(* CoDeSys 2.3.10.0 project: BC_068364(3.222)-prg__2014.10.23.prx *)
(* Libraries: standard.lbx 5.12.03 07:02:30, TcBaseBCxx50.lbx 29.3.07 05:21:36, TcSystemBCxx50.lbx*11.2.10 13:45:50, TcpIp.lib 9.1.14 12:33:22 *)

(* Task configuration *)
TASK Standard (PRIORITY := 0, INTERVAL := T#20ms);
	ADS_block();
	MAIN
END_TASK

(* Global variable list: Global_Variables *)
VAR_GLOBAL
	IN_DGU AT %I* : BOOL; (*сигнал старта дгу / IN1 на MU1.6 KL1702*)
	IN_TEMP AT %I* : INT; (*температура воздуха в гараже / IN1 на MU1.3 KL4002*)
	IN_CO2 AT %I* : INT; (*содержание СО2 в гараже / IN2 на MU1.3 KL4002*)
	OUT_START_V1 AT %Q* : BOOL; (*старт пускателя В-1 / IN1 на MU1.1 KM2642*)
	OUT_START_V2 AT %Q* : BOOL; (*старт пускателя В-2 / IN2 на MU1.1 KM2642*)
	OUT_START_V3 AT %Q* : BOOL; (*старт вентилятора в туалете Николая В-3 / IN1 на MU1.2 KM2642*)
	OUT_OUTPUT_V1 AT %Q* : INT; (*производительность В-1 / OUT1 на MU1.3 KL4002*)
	OUT_OUTPUT_V2 AT %Q* : INT; (*производительность В-2 / OUT2 на MU1.3 KL4002*)
	Ads_Udp_send_Stack : ARRAY [1..7] OF INT; (*информационный массив для передачи по ADS*)
	Ads_Udp_receive_Stack : ARRAY [1..7] OF INT; (*информационный массив для получения по ADS*)
	Ads_Udp_empty_Stack : ARRAY [1..7] OF INT := 0;
	Garage_OG10_11: BOOL := FALSE;
	Garage AT %MB10 : BOOL;

	var1 : BOOL;
	var2: BOOL;
	var3 : BOOL;
END_VAR

(* Global variable list: TwinCAT_Configuration *)
(* Generated automatically by TwinCAT - (read only) *)
VAR_CONFIG
	.IN_DGU AT %IX8.0 : BOOL;	(*  ~ {LinkedWith:TIID^Device 2 (BX-BK)^BX KBus-Device^Term 7 (KL1702)^Channel 1^Input} *)
	.IN_TEMP AT %IB12 : INT;	(*  ~ {LinkedWith:TIID^Device 2 (BX-BK)^BX KBus-Device^Term 4 (KL3062)^Channel 1^Data In} *)
	.IN_CO2 AT %IB14 : INT;	(*  ~ {LinkedWith:TIID^Device 2 (BX-BK)^BX KBus-Device^Term 4 (KL3062)^Channel 2^Data In} *)
	.OUT_START_V1 AT %QX8.0 : BOOL;	(*  ~ {LinkedWith:TIID^Device 2 (BX-BK)^BX KBus-Device^Term 2 (KM2642)^Channel 1^Output} *)
	.OUT_START_V2 AT %QX8.1 : BOOL;	(*  ~ {LinkedWith:TIID^Device 2 (BX-BK)^BX KBus-Device^Term 2 (KM2642)^Channel 2^Output} *)
	.OUT_START_V3 AT %QX8.2 : BOOL;	(*  ~ {LinkedWith:TIID^Device 2 (BX-BK)^BX KBus-Device^Term 3 (KM2642)^Channel 1^Output} *)
	.OUT_OUTPUT_V1 AT %QB12 : INT;	(*  ~ {LinkedWith:TIID^Device 2 (BX-BK)^BX KBus-Device^Term 5 (KL4002)^Channel 1^Data Out} *)
	.OUT_OUTPUT_V2 AT %QB14 : INT;	(*  ~ {LinkedWith:TIID^Device 2 (BX-BK)^BX KBus-Device^Term 5 (KL4002)^Channel 2^Data Out} *)
END_VAR

(* POU ADS_block, CFC *)
PROGRAM ADS_block
VAR
	Timer1: TON;
	ADSreadcxbc: ADSREAD;
	ADSwritecxbc: ADSWRITE;
	ADSreadcxbc2: ADSREAD;
	Timer2: TON;
END_VAR
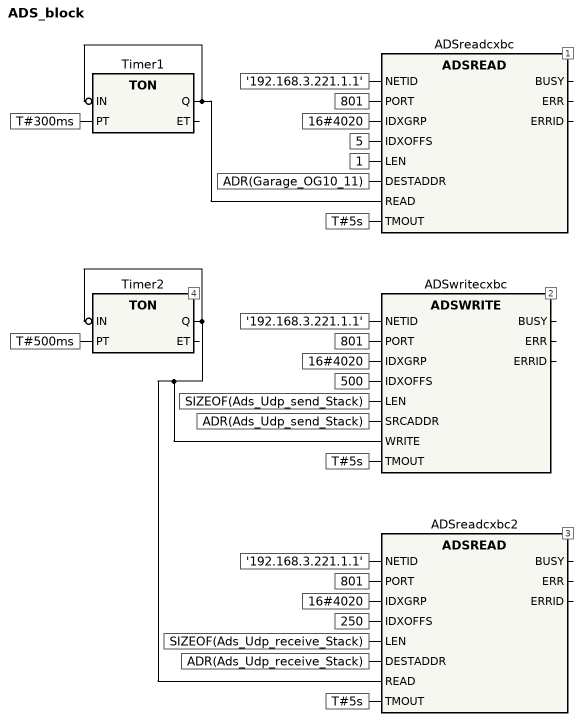
_CFC_ (* Continuous Function Chart, elements in execution order *)
#0 Timer1:TON(IN: NOT #0.Q, PT: T#300ms)
#1 ADSreadcxbc:ADSREAD(NETID: '192.168.3.221.1.1', PORT: 801, IDXGRP: 16#4020, IDXOFFS: 5, LEN: 1, DESTADDR: ADR(Garage_OG10_11), READ: #0.Q, TMOUT: T#5s)
#2 ADSwritecxbc:ADSWRITE(NETID: '192.168.3.221.1.1', PORT: 801, IDXGRP: 16#4020, IDXOFFS: 500, LEN: SIZEOF(Ads_Udp_send_Stack), SRCADDR: ADR(Ads_Udp_send_Stack), WRITE: #4.Q, TMOUT: T#5s)
#3 ADSreadcxbc2:ADSREAD(NETID: '192.168.3.221.1.1', PORT: 801, IDXGRP: 16#4020, IDXOFFS: 250, LEN: SIZEOF(Ads_Udp_receive_Stack), DESTADDR: ADR(Ads_Udp_receive_Stack), READ: #4.Q, TMOUT: T#5s)
#4 Timer2:TON(IN: NOT #4.Q, PT: T#500ms)
_END_CFC_
(* the same logic as Structured Text *)
Timer1(IN := NOT Timer1.Q, PT := T#300ms);
ADSreadcxbc(NETID := '192.168.3.221.1.1', PORT := 801, IDXGRP := 16#4020, IDXOFFS := 5, LEN := 1, DESTADDR := ADR(Garage_OG10_11), READ := Timer1.Q, TMOUT := T#5s);
ADSwritecxbc(NETID := '192.168.3.221.1.1', PORT := 801, IDXGRP := 16#4020, IDXOFFS := 500, LEN := SIZEOF(Ads_Udp_send_Stack), SRCADDR := ADR(Ads_Udp_send_Stack), WRITE := Timer2.Q, TMOUT := T#5s);
ADSreadcxbc2(NETID := '192.168.3.221.1.1', PORT := 801, IDXGRP := 16#4020, IDXOFFS := 250, LEN := SIZEOF(Ads_Udp_receive_Stack), DESTADDR := ADR(Ads_Udp_receive_Stack), READ := Timer2.Q, TMOUT := T#5s);
Timer2(IN := NOT Timer2.Q, PT := T#500ms);
END_PROGRAM

(* POU MAIN, ST *)
PROGRAM MAIN
VAR
	FirstCycle : BOOL := TRUE;
	CO2_LIMIT : INT := 8500; (*граница срабатывания датчика СО2*)
	CO2_DELTA : INT := 500; (*дисперсия*)
	PROD_V1 : INT := 32767; (*производительности В-1 при включении*)
	PROD_V2 : INT := 32767; (*производительности В-2 при включении*)
(*
	TEMP_CO2_MAX : INT;
	TEMP_CO2_MIN : INT := 32767;
*)
	k: INT;
	Rec_Not_Empty: BOOL;
	TP1: TP;
	TP2: TP;
	TP3: TP;
	TP4: TP;
	TP5: TP;
	TP6: TP;
END_VAR
OUT_OUTPUT_V1 := PROD_V1;
OUT_OUTPUT_V2 := PROD_V2;
Rec_Not_Empty := FALSE;
TP1( IN := IN_DGU, PT := T#500ms, Q => , ET =>);
TP2( IN := NOT(IN_DGU), PT := T#500ms, Q => , ET =>);
TP3( IN := IN_CO2 > CO2_LIMIT, PT := T#500ms, Q => , ET =>);
TP4( IN := IN_CO2 < CO2_LIMIT - CO2_DELTA, PT := T#500ms, Q => , ET =>);
TP5( IN := Garage_OG10_11, PT := T#500ms, Q => , ET =>);
TP6( IN := NOT(Garage_OG10_11), PT := T#500ms, Q => , ET =>);

IF TP1.Q THEN
	OUT_START_V2 := TRUE;
	OUT_OUTPUT_V2 := PROD_V2; (* старт вентилятора и производительность на максимум*)
	Ads_Udp_send_Stack[1] := 1;
	Ads_Udp_send_Stack[3] := 1;
END_IF;
IF TP2.Q THEN
	OUT_START_V2 := FALSE;
	OUT_OUTPUT_V2 := 0; (* старт вентилятора и производительность на максимум*)
	Ads_Udp_send_Stack[1] := 0;
	Ads_Udp_send_Stack[3] := 0;
END_IF;

IF TP3.Q THEN (*включение приточно-вытяжной венлиляции по сигналу загазованности*)
	OUT_START_V1 := TRUE;
	OUT_OUTPUT_V1 := PROD_V1; (* старт вентилятора и производительность на максимум*)
	Ads_Udp_send_Stack[2] := 1;
END_IF;
IF TP4.Q THEN (*выключение приточно-вытяжной венлиляции по сигналу загазованности*)
	OUT_START_V1 := FALSE;
	OUT_OUTPUT_V1 := 0;
	Ads_Udp_send_Stack[2] := 0;
END_IF;

IF TP5.Q THEN (*включение вытяжки в туалете управляющего по включению света*)
	OUT_START_V3 := TRUE;
	Ads_Udp_send_Stack[4] := 1;
END_IF;
IF TP6.Q THEN
	OUT_START_V3 := FALSE;
	Ads_Udp_send_Stack[4] := 0;
END_IF;

Ads_Udp_send_Stack[7] := IN_CO2;
Ads_Udp_send_Stack[5] := OUT_OUTPUT_V1;
Ads_Udp_send_Stack[6] := OUT_OUTPUT_V2;

FOR k := 2 TO 6 DO
IF (Ads_Udp_receive_Stack[k] = Ads_Udp_empty_Stack[k]) THEN
Rec_Not_Empty := (Rec_Not_Empty OR FALSE);
ELSE
Rec_Not_Empty := (Rec_Not_Empty OR TRUE);
END_IF;
END_FOR;

IF(Rec_Not_Empty) THEN
	IF(Ads_Udp_receive_Stack[2] = 1) THEN OUT_START_V1 := TRUE; END_IF;
	IF(Ads_Udp_receive_Stack[2] = 0) THEN OUT_START_V1 := FALSE; END_IF;
	OUT_OUTPUT_V1 := Ads_Udp_receive_Stack[5];
	Ads_Udp_send_Stack[5] := Ads_Udp_receive_Stack[5];
	Ads_Udp_send_Stack[2] := Ads_Udp_receive_Stack[2];

	IF(Ads_Udp_receive_Stack[3] = 1) THEN OUT_START_V2 := TRUE; END_IF;
	IF(Ads_Udp_receive_Stack[3] = 0) THEN OUT_START_V2 := FALSE; END_IF;
	OUT_OUTPUT_V2 := Ads_Udp_receive_Stack[6];
	Ads_Udp_send_Stack[6] := Ads_Udp_receive_Stack[6];
	Ads_Udp_send_Stack[3] := Ads_Udp_receive_Stack[3];

	IF(Ads_Udp_receive_Stack[4] = 1) THEN OUT_START_V3 := TRUE; END_IF;
	IF(Ads_Udp_receive_Stack[4] = 0) THEN OUT_START_V3 := FALSE; END_IF;
	Ads_Udp_send_Stack[4] := Ads_Udp_receive_Stack[4];
	Ads_Udp_empty_Stack := Ads_Udp_receive_Stack;
END_IF;
END_PROGRAM
